(* LS Electric XG5000 project: Function_Block_Counter *)
(* PLC LSPLC *)

FUNCTION 시간검출 : ARRAY[0..5] OF WORD
VAR_INPUT
    _RTC_TIME_0 : BYTE;
    _RTC_TIME_1 : BYTE;
    _RTC_TIME_2 : BYTE;
    _RTC_TIME_3 : BYTE;
    _RTC_TIME_4 : BYTE;
    _RTC_TIME_5 : BYTE;
END_VAR

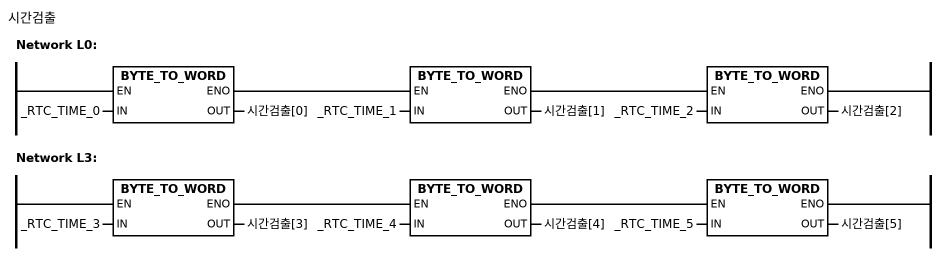
(* Rung L0 *)
시간검출[0] := BYTE_TO_WORD(_RTC_TIME_0);
시간검출[1] := BYTE_TO_WORD(_RTC_TIME_1);
시간검출[2] := BYTE_TO_WORD(_RTC_TIME_2);
(* Rung L3 *)
시간검출[3] := BYTE_TO_WORD(_RTC_TIME_3);
시간검출[4] := BYTE_TO_WORD(_RTC_TIME_4);
시간검출[5] := BYTE_TO_WORD(_RTC_TIME_5);
END_FUNCTION

FUNCTION_BLOCK 사칙연산
VAR_INPUT
    input1 : REAL;
    input2 : REAL;
END_VAR
VAR_OUTPUT
    result1 : REAL;
    result2 : REAL;
    result3 : REAL;
    resut4 : REAL;
END_VAR

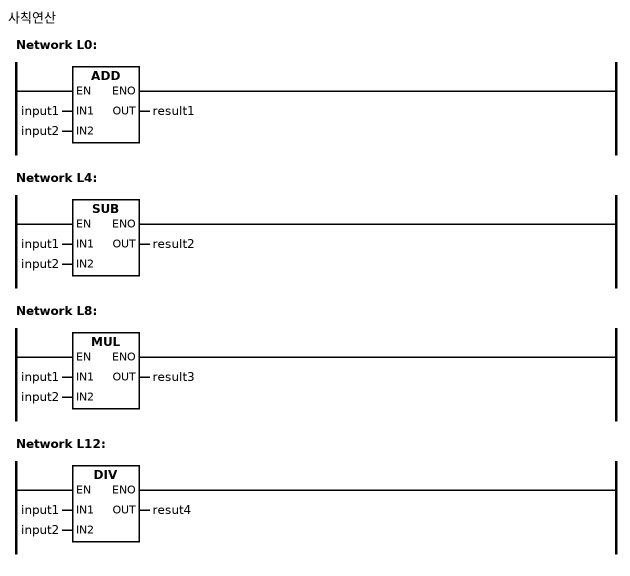
(* Rung L0 *)
result1 := input1 + input2;
(* Rung L4 *)
result2 := input1 - input2;
(* Rung L8 *)
result3 := input1 * input2;
(* Rung L12 *)
resut4 := input1 / input2;
END_FUNCTION_BLOCK

FUNCTION PITA : REAL
VAR_INPUT
    uderline : REAL;
    height : REAL;
END_VAR
VAR
    height_square : REAL;
    square : REAL;
    uderline_square : REAL;
END_VAR

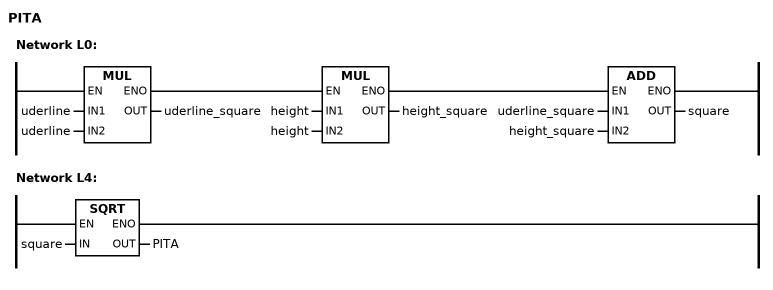
(* Rung L0 *)
uderline_square := uderline * uderline;
height_square := height * height;
square := uderline_square + height_square;
(* Rung L4 *)
PITA := SQRT(square);
END_FUNCTION

FUNCTION_BLOCK Practice
VAR_INPUT
    FL : BOOL;
    NFL : BOOL;
    OFF : BOOL;
END_VAR
VAR_OUTPUT
    LA1 : BOOL;
    LA2 : BOOL;
END_VAR
VAR
    t1 : TP;
END_VAR

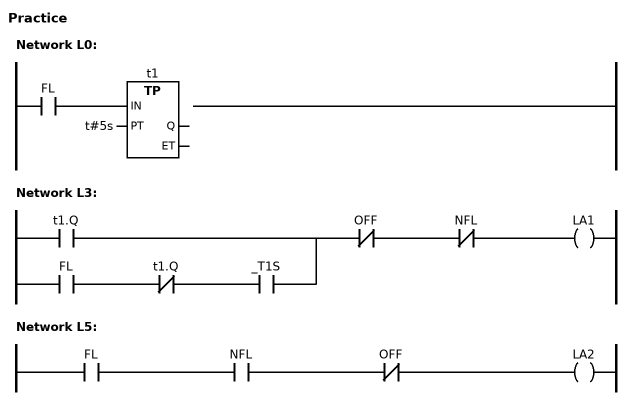
(* Rung L0 *)
t1(IN := FL, PT := t#5s);
(* Rung L3 *)
LA1 := (t1.Q OR (FL AND NOT t1.Q AND _T1S)) AND NOT OFF AND NOT NFL;
(* Rung L5 *)
LA2 := FL AND NFL AND NOT OFF;
END_FUNCTION_BLOCK

PROGRAM NewProgram (* task: 스캔 프로그램 *)
VAR
    A : REAL;
    B : REAL;
    C1 : CTU_INT;
    C2 : CTD_INT;
    C3 : CTUD_INT;
    C4 : CTD_INT;
    eqaul : BOOL;
    LD_ON : BOOL;
    LT1 : BOOL;
    LT2 : BOOL;
    P1 : Practice;
    TEST1 : 사칙연산;
    trigger : BOOL;
    램프1 : BOOL;
    램프2 : BOOL;
    램프3 : BOOL;
    램프4 : BOOL;
    램프5 : BOOL;
    리셋 : BOOL;
    스위치1 : BOOL;
    스위치2 : BOOL;
    스위치3 : BOOL;
    시간검출 : ARRAY[0..5] OF WORD;
END_VAR

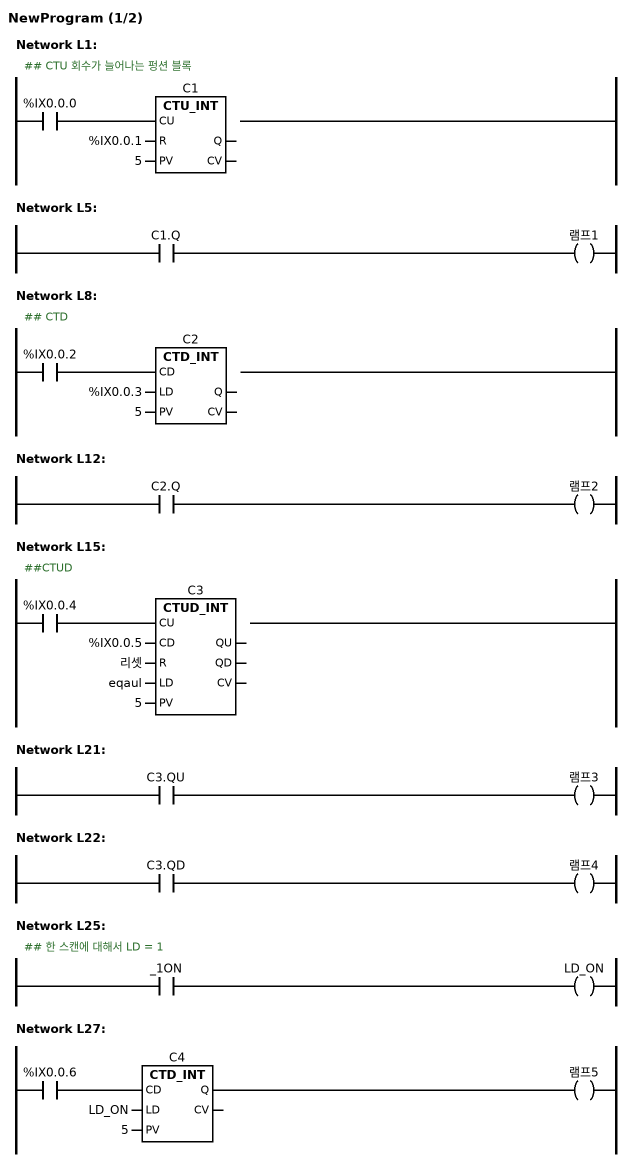
(* ## CTU 회수가 늘어나는 펑션 블록 *)
(* Rung L1 *)
C1(CU := %IX0.0.0, R := %IX0.0.1, PV := 5);
(* Rung L5 *)
램프1 := C1.Q;
(* ## CTD *)
(* Rung L8 *)
C2(CD := %IX0.0.2, LD := %IX0.0.3, PV := 5);
(* Rung L12 *)
램프2 := C2.Q;
(* ##CTUD *)
(* Rung L15 *)
C3(CU := %IX0.0.4, CD := %IX0.0.5, R := 리셋, LD := eqaul, PV := 5);
(* Rung L21 *)
램프3 := C3.QU;
(* Rung L22 *)
램프4 := C3.QD;
(* ## 한 스캔에 대해서 LD = 1 *)
(* Rung L25 *)
LD_ON := _1ON;
(* Rung L27 *)
C4(CD := %IX0.0.6, LD := LD_ON, PV := 5);
램프5 := C4.Q;

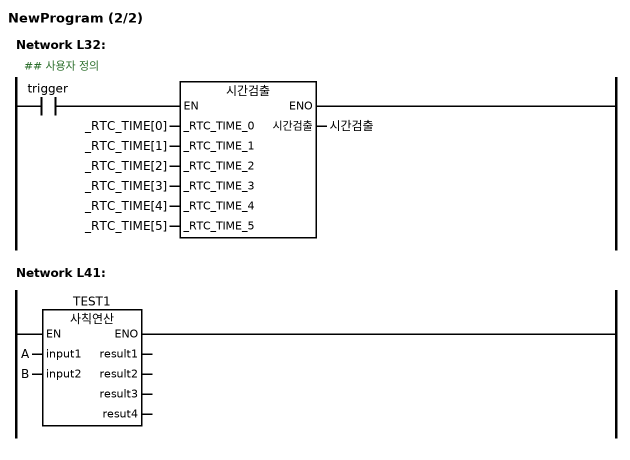
(* ## 사용자 정의 *)
(* Rung L32 *)
IF trigger THEN
    시간검출 := 시간검출(_RTC_TIME_0 := _RTC_TIME[0], _RTC_TIME_1 := _RTC_TIME[1], _RTC_TIME_2 := _RTC_TIME[2], _RTC_TIME_3 := _RTC_TIME[3], _RTC_TIME_4 := _RTC_TIME[4], _RTC_TIME_5 := _RTC_TIME[5]);
END_IF;
(* Rung L41 *)
TEST1(input1 := A, input2 := B);
END_PROGRAM

PROGRAM TEST (* task: 스캔 프로그램 *)
VAR
    A : REAL;
    B : REAL;
    C4 : CTD_INT;
    input : BOOL;
    LD_ON : BOOL;
    LT1 : BOOL;
    LT2 : BOOL;
    P1 : Practice;
    PITA : REAL;
    result : REAL;
    램프5 : BOOL;
    스위치1 : BOOL;
    스위치2 : BOOL;
    스위치3 : BOOL;
END_VAR

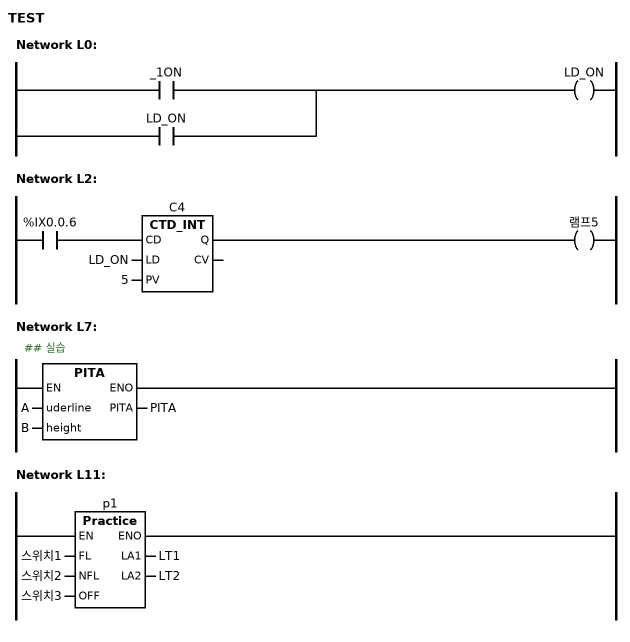
(* Rung L0 *)
LD_ON := _1ON OR LD_ON;
(* Rung L2 *)
C4(CD := %IX0.0.6, LD := LD_ON, PV := 5);
램프5 := C4.Q;
(* ## 실습 *)
(* Rung L7 *)
PITA := PITA(uderline := A, height := B);
(* Rung L11 *)
p1(FL := 스위치1, NFL := 스위치2, OFF := 스위치3, LA1 => LT1, LA2 => LT2);
END_PROGRAM